KUKA KRL program: perfil_livre.src

&ACCESS RVP
&REL 1
&PARAM TEMPLATE = C:\KRC\Roboter\Template\ExpertVorgabe
&PARAM EDITMASK = *
DEF perfil_livre( )


;FOLD ; FIM DO PROCESSO DE SOLDAGEM;%{PE}%R 4.1.16,%MKUKATPBASIS,%CCOMMENT,%VNORMAL,%P 2:FIM DO PROCESSO DE SOLDAGEM
;ENDFOLD
;FOLD PULSE 3380 'Perfil Livre Estacao' State=TRUE Time=3 sec;%{PE}%R 8.2.20,%MKUKATPBASIS,%COUT,%VPULSE,%P 2:3380, 3:Perfil Livre Estacao, 5:TRUE, 6:, 8:3
PULSE($OUT[3380], TRUE,3)
;ENDFOLD

END
